Yaskawa INFORM job: small_pipe_bent_cylinder_program.JBI

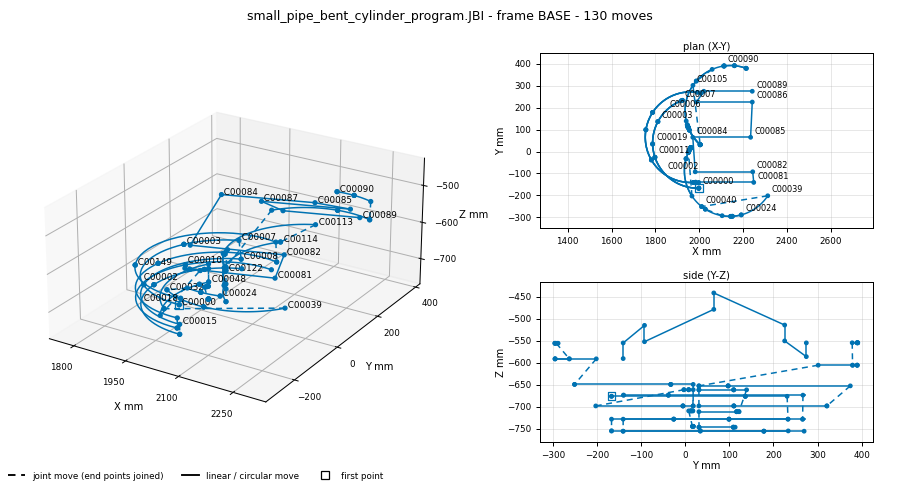
[picture p0: tool path of small_pipe_bent_cylinder_program.JBI in frame BASE, 130 of 181 moves have a stored position in this frame; points joined in program order, loops and branches not executed]
/JOB
//NAME small_pipe_bent_cylinder_program
//POS
///NPOS 170,0,170,0,0,0
///TOOL 0
///POSTYPE BASE
///RECTAN
///RCONF 0,0,0,0,0,0,0,0,0,0,0,0,0,0,0,0,0,0,0,0,0,0,0,0
C00000=1997.278396,-167.232440,-676.102460,175.000000,-60.000000,91.049110
C00001=1997.278396,-167.232440,-676.102460,175.000000,-60.000000,91.049110
C00002=1838.843025,-97.618124,-676.102460,175.000000,-60.000000,41.510842
C00003=1811.126382,136.185689,-676.102460,-175.000000,-60.000000,-27.989509
C00004=1811.126382,136.185689,-676.102460,-175.000000,-60.000000,-27.989509
C00005=1811.126382,136.185689,-676.102460,-175.000000,-60.000000,-27.989509
C00006=1846.681761,184.514776,-676.102460,175.000000,-60.000000,-44.693817
C00007=1916.740566,230.994572,-676.102460,175.000000,-60.000000,-68.182429
C00008=1921.895510,232.978673,-727.915460,175.000000,-60.000000,-69.714856
C00009=1921.895510,232.978673,-727.915460,175.000000,-60.000000,-69.714856
C00010=1811.911109,137.647989,-727.915460,175.000000,-60.000000,-28.449911
C00011=1797.607783,-26.168862,-727.915460,175.000000,-60.000000,18.469899
C00012=1797.607783,-26.168862,-727.915460,175.000000,-60.000000,18.469899
C00013=1797.607783,-26.168862,-727.915460,175.000000,-60.000000,18.469899
C00014=1877.955426,-131.922928,-727.915460,175.000000,-60.000000,55.982289
C00015=1997.836508,-167.221466,-727.915460,-175.000000,-60.000000,91.203974
C00016=1997.468714,-167.228868,-754.631960,175.000000,-60.000000,91.101918
C00017=1997.468714,-167.228868,-754.631960,175.000000,-60.000000,91.101918
C00018=1812.764618,-60.686505,-754.631960,-175.000000,-60.000000,28.943039
C00019=1787.034023,34.102385,-754.631960,175.000000,-60.000000,5.000000
C00020=1787.034023,34.102385,-754.631960,175.000000,-60.000000,5.000000
C00021=1787.034023,34.102385,-754.631960,175.000000,-60.000000,5.000000
C00022=1853.105007,190.731967,-754.631960,-175.000000,-60.000000,-47.174000
C00023=1923.294494,233.490035,-754.631960,175.000000,-60.000000,-70.128084
C00024=2191.004980,-288.807992,-555.873000,-75.326300,-90.000000,5.000000
C00025=2191.004980,-288.807992,-555.873000,-75.326300,-90.000000,5.000000
C00026=2166.443499,-293.672274,-555.873000,-82.269313,-89.999999,5.000000
C00027=2142.770132,-295.509960,-555.873000,-88.853121,-90.000000,5.000000
C00028=2142.770132,-295.509960,-555.873000,-88.853121,-90.000000,5.000000
C00029=2142.770132,-295.509960,-555.873000,-88.853121,-90.000000,5.000000
C00030=2128.051191,-295.280462,-555.873000,-92.933445,-90.000000,5.000000
C00031=2103.868540,-292.607859,-555.873000,-99.679728,-90.000000,5.000000
C00032=2027.192459,-262.947654,-591.183000,-122.615680,-90.000000,5.000000
C00033=2027.192459,-262.947654,-591.183000,-122.615680,-90.000000,5.000000
C00034=2135.960585,-295.534121,-591.183000,-90.740304,-90.000000,5.000000
C00035=2150.262350,-295.223994,-591.183000,-86.775224,-89.999999,5.000000
C00036=2150.262350,-295.223994,-591.183000,-86.775224,-89.999999,5.000000
C00037=2150.262350,-295.223994,-591.183000,-86.775224,-89.999999,5.000000
C00038=2166.811995,-293.621912,-591.183000,-82.166245,-89.999999,5.000000
C00039=2311.749560,-201.833036,-591.183000,-33.141642,-90.000000,5.000000
C00040=2010.510884,-251.068811,-649.128500,-128.293165,-90.000000,5.000000
C00041=2010.510884,-251.068811,-649.128500,-128.293165,-90.000000,5.000000
C00042=1935.359523,-51.029220,-649.128500,169.473800,-90.000000,5.000000
C00043=1939.589032,-32.869333,-649.128500,164.304824,-90.000000,5.000000
C00044=1939.589032,-32.869333,-649.128500,164.304824,-90.000000,5.000000
C00045=1939.589032,-32.869333,-649.128500,164.304824,-90.000000,5.000000
C00046=1957.226392,10.388570,-649.128500,151.331203,-89.999999,5.000000
C00047=1961.553026,17.921169,-649.128500,148.923719,-90.000000,5.000000
C00048=1961.513001,17.854728,-697.952500,148.945214,-90.000000,5.000000
C00049=1961.513001,17.854728,-697.952500,148.945214,-90.000000,5.000000
C00050=1954.687250,5.596468,-697.952500,152.834152,-90.000000,5.000000
C00051=1949.525612,-5.222895,-697.952500,156.156648,-89.999999,5.000000
C00052=1949.525612,-5.222895,-697.952500,156.156648,-89.999999,5.000000
C00053=1949.525612,-5.222895,-697.952500,156.156648,-89.999999,5.000000
C00054=1942.719058,-22.735882,-697.952500,161.365372,-90.000000,5.000000
C00055=1966.290930,-203.013762,-697.952500,-146.466703,-89.999999,5.000000
C00056=1950.477237,-3.102014,-661.219960,175.000000,-60.000000,-24.487554
C00057=1950.477237,-3.102014,-661.219960,175.000000,-60.000000,-24.487554
C00058=1954.296214,4.830560,-661.219960,175.000000,-60.000000,-26.927533
C00059=1955.807104,7.747516,-661.219960,175.000000,-60.000000,-27.837902
C00060=1955.807104,7.747516,-661.219960,175.000000,-60.000000,-27.837902
C00061=1955.807104,7.747516,-661.219960,175.000000,-60.000000,-27.837902
C00062=1957.984607,11.762850,-661.219960,-175.000000,-60.000000,-29.103762
C00063=1961.594436,17.989848,-661.219960,175.000000,-60.000000,-31.098506
C00064=1961.041445,17.067677,-709.170460,-175.000000,-60.000000,-30.800524
C00065=1961.041445,17.067677,-709.170460,-175.000000,-60.000000,-30.800524
C00066=1959.883350,15.100383,-709.170460,175.000000,-60.000000,-30.167887
C00067=1958.606302,12.871609,-709.170460,-175.000000,-60.000000,-29.456031
C00068=1958.606302,12.871609,-709.170460,-175.000000,-60.000000,-29.456031
C00069=1958.606302,12.871609,-709.170460,-175.000000,-60.000000,-29.456031
C00070=1957.181566,10.306542,-709.170460,175.000000,-60.000000,-28.642893
C00071=1955.815325,7.763083,-709.170460,175.000000,-60.000000,-27.842781
C00072=1960.544274,16.229194,-744.259460,175.000000,-60.000000,-30.530384
C00073=1960.544274,16.229194,-744.259460,175.000000,-60.000000,-30.530384
C00074=1961.394939,17.658418,-744.259460,175.000000,-60.000000,-30.991303
C00075=1961.516354,17.860295,-744.259460,-175.000000,-60.000000,-31.056587
C00076=1961.516354,17.860295,-744.259460,-175.000000,-60.000000,-31.056587
C00077=1961.516354,17.860295,-744.259460,-175.000000,-60.000000,-31.056587
C00078=1961.548988,17.914468,-744.259460,175.000000,-60.000000,-31.074113
C00079=1961.587333,17.978071,-744.259460,-175.000000,-60.000000,-31.094694
C00080=1997.106118,-140.836519,-590.507414,175.000000,-60.000000,88.905037
C00081=2247.831316,-140.836514,-555.079479,175.000000,-60.000000,88.905037
C00082=2243.251187,-92.475577,-515.246497,175.000000,-50.392050,83.285154
C00083=1981.122973,-92.475582,-552.285699,175.000000,-50.392050,83.285154
C00084=1970.172616,64.700642,-478.919299,-175.000000,-8.041830,-5.000000
C00085=2233.568437,64.700647,-441.700981,-175.000000,-8.041830,-5.000000
C00086=2241.166186,225.446172,-514.516668,175.000000,-50.032545,-83.198519
C00087=1986.564308,225.446167,-550.492385,175.000000,-50.032545,-83.198519
C00088=2020.405221,274.512312,-586.146765,-175.000000,-60.000000,-88.762425
C00089=2241.157658,274.512316,-554.954037,-175.000000,-60.000000,-88.762425
C00090=2110.929813,389.536129,-554.742000,98.561467,-89.999999,5.000000
C00091=2110.929813,389.536129,-554.742000,98.561467,-89.999999,5.000000
C00092=2129.010759,391.449702,-554.742000,93.521201,-90.000000,5.000000
C00093=2159.777611,391.048975,-554.742000,84.986368,-90.000000,5.000000
C00094=2159.777611,391.048975,-554.742000,84.986368,-90.000000,5.000000
C00095=2159.777611,391.048975,-554.742000,84.986368,-90.000000,5.000000
C00096=2188.593596,386.453911,-554.742000,76.893159,-90.000000,5.000000
C00097=2214.588922,378.569027,-554.742000,69.359716,-90.000000,5.000000
C00098=2212.323915,379.407132,-605.573500,70.028999,-90.000000,5.000000
C00099=2212.323915,379.407132,-605.573500,70.028999,-90.000000,5.000000
C00100=2179.455995,388.365054,-605.573500,79.480417,-89.999999,5.000000
C00101=2113.453531,389.900169,-605.573500,97.854842,-89.999999,5.000000
C00102=2113.453531,389.900169,-605.573500,97.854842,-89.999999,5.000000
C00103=2113.453531,389.900169,-605.573500,97.854842,-89.999999,5.000000
C00104=1974.871823,307.201460,-605.573500,143.798484,-89.999999,5.000000
C00105=1970.787320,301.415623,-605.573500,145.761255,-89.999999,5.000000
C00106=2003.875571,30.983783,-652.470000,-131.809933,-89.999999,5.000000
C00107=2003.875571,30.983783,-652.470000,-131.809933,-89.999999,5.000000
C00108=1974.804817,63.066782,-652.470000,-143.829936,-90.000000,5.000000
C00109=1954.545876,97.246264,-652.470000,-154.857730,-90.000000,5.000000
C00110=1954.545876,97.246264,-652.470000,-154.857730,-90.000000,5.000000
C00111=1954.545876,97.246264,-652.470000,-154.857730,-90.000000,5.000000
C00112=1938.535751,146.788290,-652.470000,-169.324495,-90.000000,5.000000
C00113=2058.360437,374.295299,-652.470000,113.774226,-90.000000,5.000000
C00114=1986.012187,321.120540,-697.941500,138.856308,-90.000000,5.000000
C00115=1986.012187,321.120540,-697.941500,138.856308,-90.000000,5.000000
C00116=1938.961467,144.595121,-697.941500,-168.705369,-89.999999,5.000000
C00117=1949.010453,110.164814,-697.941500,-158.753322,-90.000000,5.000000
C00118=1949.010453,110.164814,-697.941500,-158.753322,-90.000000,5.000000
C00119=1949.010453,110.164814,-697.941500,-158.753322,-90.000000,5.000000
C00120=1973.007824,65.563531,-697.941500,-144.682428,-90.000000,5.000000
C00121=2003.929390,30.935663,-697.941500,-131.789926,-90.000000,5.000000
C00122=2003.940281,30.925929,-661.417960,-175.000000,-60.000000,48.214122
C00123=2003.940281,30.925929,-661.417960,-175.000000,-60.000000,48.214122
C00124=1974.995438,62.806473,-661.417960,175.000000,-60.000000,36.259476
C00125=1949.158513,109.785123,-661.417960,175.000000,-60.000000,21.359616
C00126=1949.158513,109.785123,-661.417960,175.000000,-60.000000,21.359616
C00127=1949.158513,109.785123,-661.417960,175.000000,-60.000000,21.359616
C00128=1944.366245,123.427162,-661.417960,175.000000,-60.000000,17.351788
C00129=1940.142664,139.074476,-661.417960,175.000000,-60.000000,12.859207
C00130=1944.893966,121.762939,-711.008460,175.000000,-60.000000,17.835617
C00131=1944.893966,121.762939,-711.008460,175.000000,-60.000000,17.835617
C00132=1945.651536,119.455002,-711.008460,175.000000,-60.000000,18.508779
C00133=1946.669721,116.488456,-711.008460,175.000000,-60.000000,19.377962
C00134=1946.669721,116.488456,-711.008460,175.000000,-60.000000,19.377962
C00135=1946.669721,116.488456,-711.008460,175.000000,-60.000000,19.377962
C00136=1949.065623,110.023075,-711.008460,-175.000000,-60.000000,21.288827
C00137=2003.876794,30.982689,-711.008460,175.000000,-60.000000,48.190522
C00138=2003.665373,31.172045,-746.186960,175.000000,-60.000000,48.111868
C00139=2003.665373,31.172045,-746.186960,175.000000,-60.000000,48.111868
C00140=2000.969896,33.632825,-746.186960,-175.000000,-60.000000,47.100410
C00141=1949.470303,108.992688,-746.186960,175.000000,-60.000000,21.595605
C00142=1949.470303,108.992688,-746.186960,175.000000,-60.000000,21.595605
C00143=1949.470303,108.992688,-746.186960,175.000000,-60.000000,21.595605
C00144=1948.958546,110.298453,-746.186960,175.000000,-60.000000,21.206948
C00145=1947.876843,113.148369,-746.186960,175.000000,-60.000000,20.362185
C00146=1983.234517,-139.978039,-673.512960,175.000000,-60.000000,96.462395
C00147=1983.234517,-139.978039,-673.512960,175.000000,-60.000000,96.462395
C00148=1870.116709,-120.710295,-673.512960,175.000000,-60.000000,64.204382
C00149=1781.272794,-38.270691,-673.512960,-175.000000,-60.000000,30.078215
C00150=1781.272794,-38.270691,-673.512960,-175.000000,-60.000000,30.078215
C00151=1781.272794,-38.270691,-673.512960,-175.000000,-60.000000,30.078215
C00152=1753.463632,64.477689,-673.512960,-175.000000,-60.000000,5.000000
C00153=2004.632704,266.881720,-673.512960,175.000000,-60.000000,-102.483621
C00154=2007.825450,266.148253,-727.995460,175.000000,-60.000000,-103.392449
C00155=2007.825450,266.148253,-727.995460,175.000000,-60.000000,-103.392449
C00156=1868.871861,250.577620,-727.995460,175.000000,-60.000000,-63.820183
C00157=1756.260219,99.117624,-727.995460,175.000000,-60.000000,-9.441975
C00158=1756.260219,99.117624,-727.995460,175.000000,-60.000000,-9.441975
C00159=1756.260219,99.117624,-727.995460,175.000000,-60.000000,-9.441975
C00160=1813.751923,-80.598786,-727.995460,175.000000,-60.000000,44.921169
C00161=1973.552217,-140.844520,-727.995460,175.000000,-60.000000,93.765303
C00162=1972.723630,-140.897378,-755.256960,175.000000,-60.000000,93.534965
C00163=1972.723630,-140.897378,-755.256960,175.000000,-60.000000,93.534965
C00164=1786.599767,-46.965958,-755.256960,175.000000,-60.000000,32.907476
C00165=1787.114010,178.230813,-755.256960,-175.000000,-60.000000,-33.169149
C00166=1787.114010,178.230813,-755.256960,-175.000000,-60.000000,-33.169149
C00167=1787.114010,178.230813,-755.256960,-175.000000,-60.000000,-33.169149
C00168=1864.752988,248.495219,-755.256960,-175.000000,-60.000000,-62.539743
C00169=1990.312446,269.526315,-755.256960,175.000000,-60.000000,-98.442814
///POSTYPE PULSE
///PULSE
EX00000=102400.0
EX00001=152576.0
EX00002=196608.0
EX00003=233472.0
EX00004=271360.0
///POSTYPE PULSE
///PULSE
EC00000=102400.0
EC00001=102400.0
EC00002=102400.0
EC00003=102400.0
EC00004=102400.0
EC00005=102400.0
EC00006=102400.0
EC00007=102400.0
EC00008=102400.0
EC00009=102400.0
EC00010=102400.0
EC00011=102400.0
EC00012=102400.0
EC00013=102400.0
EC00014=102400.0
EC00015=102400.0
EC00016=102400.0
EC00017=102400.0
EC00018=102400.0
EC00019=102400.0
EC00020=102400.0
EC00021=102400.0
EC00022=102400.0
EC00023=102400.0
EC00024=152576.0
EC00025=152576.0
EC00026=152576.0
EC00027=152576.0
EC00028=152576.0
EC00029=152576.0
EC00030=152576.0
EC00031=152576.0
EC00032=152576.0
EC00033=152576.0
EC00034=152576.0
EC00035=152576.0
EC00036=152576.0
EC00037=152576.0
EC00038=152576.0
EC00039=152576.0
EC00040=152576.0
EC00041=152576.0
EC00042=152576.0
EC00043=152576.0
EC00044=152576.0
EC00045=152576.0
EC00046=152576.0
EC00047=152576.0
EC00048=152576.0
EC00049=152576.0
EC00050=152576.0
EC00051=152576.0
EC00052=152576.0
EC00053=152576.0
EC00054=152576.0
EC00055=152576.0
EC00056=152576.0
EC00057=152576.0
EC00058=152576.0
EC00059=152576.0
EC00060=152576.0
EC00061=152576.0
EC00062=152576.0
EC00063=152576.0
EC00064=152576.0
EC00065=152576.0
EC00066=152576.0
EC00067=152576.0
EC00068=152576.0
EC00069=152576.0
EC00070=152576.0
EC00071=152576.0
EC00072=152576.0
EC00073=152576.0
EC00074=152576.0
EC00075=152576.0
EC00076=152576.0
EC00077=152576.0
EC00078=152576.0
EC00079=152576.0
EC00080=196608.0
EC00081=196608.0
EC00082=196608.0
EC00083=196608.0
EC00084=196608.0
EC00085=196608.0
EC00086=196608.0
EC00087=196608.0
EC00088=196608.0
EC00089=196608.0
EC00090=233472.0
EC00091=233472.0
EC00092=233472.0
EC00093=233472.0
EC00094=233472.0
EC00095=233472.0
EC00096=233472.0
EC00097=233472.0
EC00098=233472.0
EC00099=233472.0
EC00100=233472.0
EC00101=233472.0
EC00102=233472.0
EC00103=233472.0
EC00104=233472.0
EC00105=233472.0
EC00106=233472.0
EC00107=233472.0
EC00108=233472.0
EC00109=233472.0
EC00110=233472.0
EC00111=233472.0
EC00112=233472.0
EC00113=233472.0
EC00114=233472.0
EC00115=233472.0
EC00116=233472.0
EC00117=233472.0
EC00118=233472.0
EC00119=233472.0
EC00120=233472.0
EC00121=233472.0
EC00122=233472.0
EC00123=233472.0
EC00124=233472.0
EC00125=233472.0
EC00126=233472.0
EC00127=233472.0
EC00128=233472.0
EC00129=233472.0
EC00130=233472.0
EC00131=233472.0
EC00132=233472.0
EC00133=233472.0
EC00134=233472.0
EC00135=233472.0
EC00136=233472.0
EC00137=233472.0
EC00138=233472.0
EC00139=233472.0
EC00140=233472.0
EC00141=233472.0
EC00142=233472.0
EC00143=233472.0
EC00144=233472.0
EC00145=233472.0
EC00146=271360.0
EC00147=271360.0
EC00148=271360.0
EC00149=271360.0
EC00150=271360.0
EC00151=271360.0
EC00152=271360.0
EC00153=271360.0
EC00154=271360.0
EC00155=271360.0
EC00156=271360.0
EC00157=271360.0
EC00158=271360.0
EC00159=271360.0
EC00160=271360.0
EC00161=271360.0
EC00162=271360.0
EC00163=271360.0
EC00164=271360.0
EC00165=271360.0
EC00166=271360.0
EC00167=271360.0
EC00168=271360.0
EC00169=271360.0
//INST
///DATE 2023/08/16 14:34
///ATTR SC,RW,RJ
////FRAME BASE
///GROUP1 RB1,ST1
NOP
MOVJ P009 EX000 VJ=15.00
MOVJ C00000 EC00000 VJ=15.0
CALL JOB:SPYON
MOVC C00001 EC00001 V=150.0
MOVC C00002 EC00002 V=150.0
MOVC C00003 EC00003 V=150.0
MOVJ C00004 EC00004 VJ=15.0
MOVC C00005 EC00005 V=150.0
MOVC C00006 EC00006 V=150.0
MOVC C00007 EC00007 V=150.0
MOVJ C00008 EC00008 VJ=15.0
MOVC C00009 EC00009 V=150.0
MOVC C00010 EC00010 V=150.0
MOVC C00011 EC00011 V=150.0
MOVJ C00012 EC00012 VJ=15.0
MOVC C00013 EC00013 V=150.0
MOVC C00014 EC00014 V=150.0
MOVC C00015 EC00015 V=150.0
MOVJ C00016 EC00016 VJ=15.0
MOVC C00017 EC00017 V=150.0
MOVC C00018 EC00018 V=150.0
MOVC C00019 EC00019 V=150.0
MOVJ C00020 EC00020 VJ=15.0
MOVC C00021 EC00021 V=150.0
MOVC C00022 EC00022 V=150.0
MOVC C00023 EC00023 V=150.0
CALL JOB:SPYOF
MOVJ P009 VJ=15.00
MOVL P009 EX00000 V=150.0
MOVJ C00024 EC00024 VJ=15.0
CALL JOB:SPYON
MOVC C00025 EC00025 V=150.0
MOVC C00026 EC00026 V=150.0
MOVC C00027 EC00027 V=150.0
MOVJ C00028 EC00028 VJ=15.0
MOVC C00029 EC00029 V=150.0
MOVC C00030 EC00030 V=150.0
MOVC C00031 EC00031 V=150.0
MOVJ C00032 EC00032 VJ=15.0
MOVC C00033 EC00033 V=150.0
MOVC C00034 EC00034 V=150.0
MOVC C00035 EC00035 V=150.0
MOVJ C00036 EC00036 VJ=15.0
MOVC C00037 EC00037 V=150.0
MOVC C00038 EC00038 V=150.0
MOVC C00039 EC00039 V=150.0
MOVJ C00040 EC00040 VJ=15.0
MOVC C00041 EC00041 V=150.0
MOVC C00042 EC00042 V=150.0
MOVC C00043 EC00043 V=150.0
MOVJ C00044 EC00044 VJ=15.0
MOVC C00045 EC00045 V=150.0
MOVC C00046 EC00046 V=150.0
MOVC C00047 EC00047 V=150.0
MOVJ C00048 EC00048 VJ=15.0
MOVC C00049 EC00049 V=150.0
MOVC C00050 EC00050 V=150.0
MOVC C00051 EC00051 V=150.0
MOVJ C00052 EC00052 VJ=15.0
MOVC C00053 EC00053 V=150.0
MOVC C00054 EC00054 V=150.0
MOVC C00055 EC00055 V=150.0
MOVJ C00056 EC00056 VJ=15.0
MOVC C00057 EC00057 V=150.0
MOVC C00058 EC00058 V=150.0
MOVC C00059 EC00059 V=150.0
MOVJ C00060 EC00060 VJ=15.0
MOVC C00061 EC00061 V=150.0
MOVC C00062 EC00062 V=150.0
MOVC C00063 EC00063 V=150.0
MOVJ C00064 EC00064 VJ=15.0
MOVC C00065 EC00065 V=150.0
MOVC C00066 EC00066 V=150.0
MOVC C00067 EC00067 V=150.0
MOVJ C00068 EC00068 VJ=15.0
MOVC C00069 EC00069 V=150.0
MOVC C00070 EC00070 V=150.0
MOVC C00071 EC00071 V=150.0
MOVJ C00072 EC00072 VJ=15.0
MOVC C00073 EC00073 V=150.0
MOVC C00074 EC00074 V=150.0
MOVC C00075 EC00075 V=150.0
MOVJ C00076 EC00076 VJ=15.0
MOVC C00077 EC00077 V=150.0
MOVC C00078 EC00078 V=150.0
MOVC C00079 EC00079 V=150.0
CALL JOB:SPYOF
MOVJ P009 VJ=15.00
MOVL P009 EX00001 V=150.0
MOVJ C00080 EC00080 VJ=15.0
CALL JOB:SPYON
MOVL C00081 EC00081 V=150.0
MOVL C00082 EC00082 V=150.0
MOVL C00083 EC00083 V=150.0
MOVL C00084 EC00084 V=150.0
MOVL C00085 EC00085 V=150.0
MOVL C00086 EC00086 V=150.0
MOVL C00087 EC00087 V=150.0
MOVL C00088 EC00088 V=150.0
MOVL C00089 EC00089 V=150.0
CALL JOB:SPYOF
MOVJ P009 VJ=15.00
MOVL P009 EX00002 V=150.0
MOVJ C00090 EC00090 VJ=15.0
CALL JOB:SPYON
MOVC C00091 EC00091 V=150.0
MOVC C00092 EC00092 V=150.0
MOVC C00093 EC00093 V=150.0
MOVJ C00094 EC00094 VJ=15.0
MOVC C00095 EC00095 V=150.0
MOVC C00096 EC00096 V=150.0
MOVC C00097 EC00097 V=150.0
MOVJ C00098 EC00098 VJ=15.0
MOVC C00099 EC00099 V=150.0
MOVC C00100 EC00100 V=150.0
MOVC C00101 EC00101 V=150.0
MOVJ C00102 EC00102 VJ=15.0
MOVC C00103 EC00103 V=150.0
MOVC C00104 EC00104 V=150.0
MOVC C00105 EC00105 V=150.0
MOVJ C00106 EC00106 VJ=15.0
MOVC C00107 EC00107 V=150.0
MOVC C00108 EC00108 V=150.0
MOVC C00109 EC00109 V=150.0
MOVJ C00110 EC00110 VJ=15.0
MOVC C00111 EC00111 V=150.0
MOVC C00112 EC00112 V=150.0
MOVC C00113 EC00113 V=150.0
MOVJ C00114 EC00114 VJ=15.0
MOVC C00115 EC00115 V=150.0
MOVC C00116 EC00116 V=150.0
MOVC C00117 EC00117 V=150.0
MOVJ C00118 EC00118 VJ=15.0
MOVC C00119 EC00119 V=150.0
MOVC C00120 EC00120 V=150.0
MOVC C00121 EC00121 V=150.0
MOVJ C00122 EC00122 VJ=15.0
MOVC C00123 EC00123 V=150.0
MOVC C00124 EC00124 V=150.0
MOVC C00125 EC00125 V=150.0
MOVJ C00126 EC00126 VJ=15.0
MOVC C00127 EC00127 V=150.0
MOVC C00128 EC00128 V=150.0
MOVC C00129 EC00129 V=150.0
MOVJ C00130 EC00130 VJ=15.0
MOVC C00131 EC00131 V=150.0
MOVC C00132 EC00132 V=150.0
MOVC C00133 EC00133 V=150.0
MOVJ C00134 EC00134 VJ=15.0
MOVC C00135 EC00135 V=150.0
MOVC C00136 EC00136 V=150.0
MOVC C00137 EC00137 V=150.0
MOVJ C00138 EC00138 VJ=15.0
MOVC C00139 EC00139 V=150.0
MOVC C00140 EC00140 V=150.0
MOVC C00141 EC00141 V=150.0
MOVJ C00142 EC00142 VJ=15.0
MOVC C00143 EC00143 V=150.0
MOVC C00144 EC00144 V=150.0
MOVC C00145 EC00145 V=150.0
CALL JOB:SPYOF
MOVJ P009 VJ=15.00
MOVL P009 EX00003 V=150.0
MOVJ C00146 EC00146 VJ=15.0
CALL JOB:SPYON
MOVC C00147 EC00147 V=150.0
MOVC C00148 EC00148 V=150.0
MOVC C00149 EC00149 V=150.0
MOVJ C00150 EC00150 VJ=15.0
MOVC C00151 EC00151 V=150.0
MOVC C00152 EC00152 V=150.0
MOVC C00153 EC00153 V=150.0
MOVJ C00154 EC00154 VJ=15.0
MOVC C00155 EC00155 V=150.0
MOVC C00156 EC00156 V=150.0
MOVC C00157 EC00157 V=150.0
MOVJ C00158 EC00158 VJ=15.0
MOVC C00159 EC00159 V=150.0
MOVC C00160 EC00160 V=150.0
MOVC C00161 EC00161 V=150.0
MOVJ C00162 EC00162 VJ=15.0
MOVC C00163 EC00163 V=150.0
MOVC C00164 EC00164 V=150.0
MOVC C00165 EC00165 V=150.0
MOVJ C00166 EC00166 VJ=15.0
MOVC C00167 EC00167 V=150.0
MOVC C00168 EC00168 V=150.0
MOVC C00169 EC00169 V=150.0
CALL JOB:SPYOF
MOVJ P009 VJ=15.00
MOVL P009 EX00004 V=150.0
END
